// TIA Portal V19 export
FUNCTION_BLOCK "RH_OUT_TR"   // FB1, FBD
{ S7_Optimized_Access := 'TRUE' }
// stored: MemoryReserve 100, SetENOAutomatically false
   VAR_INPUT
      Address : HW_IO;
      GL1 : Bool;
      GL2 : Bool;
      Fwd : Bool;
      Rev : Bool;
      InterlockOk : Bool;
   END_VAR
   VAR_OUTPUT
      Speed_PV : Int;
      Status : Int;
   END_VAR
   VAR
      Frq : "RMP_BIF_FRQ_SPD";   // Device frequency converter control / Laitteen taajuusmuuttajan ohjaus
      Drive { S7_SetPoint := 'True'} : "RMP_FRQ_SPD";
      Control : "RMP_UDT_CONTROL";   // Laitteen ohjaus / Device control
      "Status.Ack" { S7_SetPoint := 'True'} : Bool;
   END_VAR
BEGIN

REGION Network 1: Device fwd request
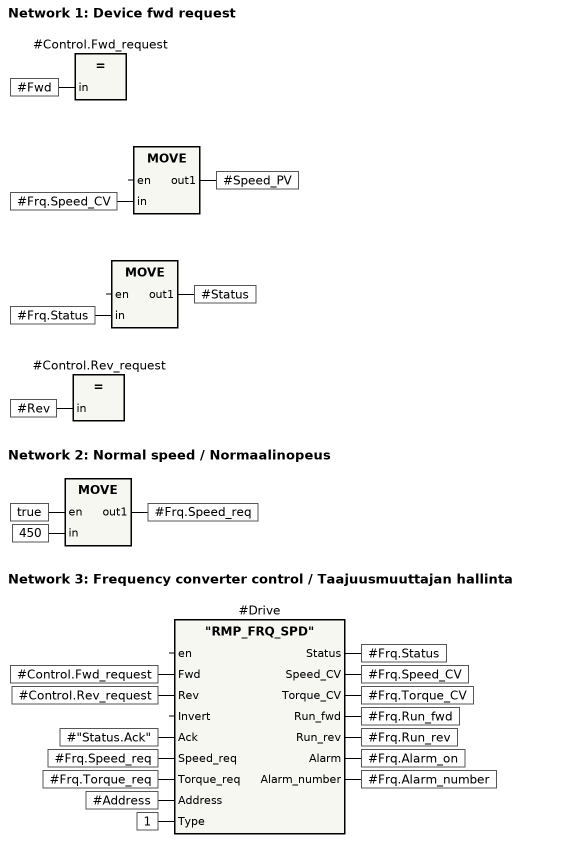
   #Control.Fwd_request := #Fwd;
   #Speed_PV := #Frq.Speed_CV;
   #Status := #Frq.Status;
   #Control.Rev_request := #Rev;
END_REGION

REGION Network 2: Normal speed / Normaalinopeus
   IF true THEN #Frq.Speed_req := 450; END_IF;
END_REGION

REGION Network 3: Frequency converter control / Taajuusmuuttajan hallinta
   #Drive(Fwd := #Control.Fwd_request,   // "RMP_FRQ_SPD"
          Rev := #Control.Rev_request,
          Ack := #"Status.Ack",
          Speed_req := #Frq.Speed_req,
          Torque_req := #Frq.Torque_req,
          Address := #Address,
          "Type" := 1,
          Status => #Frq.Status,
          Speed_CV => #Frq.Speed_CV,
          Torque_CV => #Frq.Torque_CV,
          Run_fwd => #Frq.Run_fwd,
          Run_rev => #Frq.Run_rev,
          Alarm => #Frq.Alarm_on,
          Alarm_number => #Frq.Alarm_number);
END_REGION
END_FUNCTION_BLOCK
